FUNCTION TryConvert_DATE_TO_TIME : BOOL
VAR_INPUT
	in : DATE;
	out : REFERENCE TO TIME;
END_VAR

IF in > TIME_TO_DATE(T#49D17H2M47S295MS) THEN
	RETURN;
END_IF

out := DATE_TO_TIME(in);
TryConvert_DATE_TO_TIME := TRUE;

END_FUNCTION

(* stored: Version 1.1.0.1, ProductVersion 3.1.4024.12
   POU TryConvert_DATE_TO_TIME: Id {2713f4ac-162f-4e4b-9f32-845d185859aa}, SpecialFunc None *)
